// TIA Portal project "sauc" (V13)

(* hardware
DEVICE "HMI_1"  TP700 Comfort
   slot 0: "HMI"  HMI  6AV2 124-0GC01-0AX0  13.0.1.0
   slot 1: "HMI_RT_1"  TP700 Comfort  6AV2 124-0GC01-0AX0  13.0.1.0
   slot 5: "HMI_1.IE_CP_1"  PROFINET Interface
      slot 1: "PROFINET Interface_1"  PROFINET Interface
         slot 1: "Port_1"  Port
         slot 2: "Port_2"  Port
   slot 7: "HMI_1.MPI/DP_CP_1"  MPI/DP Interface
*)

(* ===== HMI "HMI_RT_1" =====
connection "CPU224": IF1 B, SIMATIC S7 200

HMI tags "Default tag table"
   "lightSensor" : Bool, 1 s
   "openDoor" : Bool, 1 s
   "lowBob" : Bool, 1 s
   "upBob" : Bool, 1 s
   "heaterGoOn" : Bool, 1 s
   "lightGoOn" : Bool, 1 s
   "doorGoOn" : Bool, 1 s
   "ventilGoOn" : Bool, 1 s
   "valve1goOn" : Bool, 1 s
   "valve2goOn" : Bool, 1 s
   "valve3goOn" : Bool, 1 s
   "lightBySensor" : Bool, 1 s
   "lightByTime" : Bool, 1 s
   "readYear" : Byte, 1 s
   "readMonth" : Byte, 1 s
   "readDay" : Byte, 1 s
   "readHours" : Byte, 1 s
   "readMinutes" : Byte, 1 s
   "readSeconds" : Byte, 1 s
   "writeYear" : Byte, 1 s
   "writeMonth" : Byte, 1 s
   "writeDay" : Byte, 1 s
   "writeHours" : Byte, 1 s
   "writeMinutes" : Byte, 1 s
   "writeSeconds" : Byte, 1 s
   "roomTemp4ma" : Real, 1 s
   "roomTemp20ma" : Real, 1 s
   "airTemp4ma" : Real, 1 s
   "airTemp20ma" : Real, 1 s
   "humidityRoom4ma" : Real, 1 s
   "humidityRoom20ma" : Real, 1 s
   "floorTemp4ma" : Real, 1 s
   "floorTemp20ma" : Real, 1 s
   "roomTemp" : Real, 1 s
   "airTemp" : Real, 1 s
   "humidityRoom" : Real, 1 s
   "floorTemp" : Real, 1 s
   "v1_e1_on_hh" : Byte, 1 s
   "v1_e1_on_mm" : Byte, 1 s
   "v1_e1_off_hh" : Byte, 1 s
   "v1_e1_off_mm" : Byte, 1 s
   "v1_e2_on_hh" : Byte, 1 s
   "v1_e2_on_mm" : Byte, 1 s
   "v1_e2_off_hh" : Byte, 1 s
   "v1_e2_off_mm" : Byte, 1 s
   "v1_e3_on_hh" : Byte, 1 s
   "v1_e3_on_mm" : Byte, 1 s
   "v1_e3_off_hh" : Byte, 1 s
   "v1_e3_off_mm" : Byte, 1 s
   "v1_e4_on_hh" : Byte, 1 s
   "v1_e4_on_mm" : Byte, 1 s
   "v1_e4_off_hh" : Byte, 1 s
   "v1_e4_off_mm" : Byte, 1 s
   "v1_e5_on_hh" : Byte, 1 s
   "v1_e5_on_mm" : Byte, 1 s
   "v1_e5_off_hh" : Byte, 1 s
   "v1_e5_off_mm" : Byte, 1 s
   "v2_e1_on_hh" : Byte, 1 s
   "v2_e1_on_mm" : Byte, 1 s
   "v2_e1_off_hh" : Byte, 1 s
   "v2_e1_off_mm" : Byte, 1 s
   "v2_e2_on_hh" : Byte, 1 s
   "v2_e2_on_mm" : Byte, 1 s
   "v2_e2_off_hh" : Byte, 1 s
   "v2_e2_off_mm" : Byte, 1 s
   "v2_e3_on_hh" : Byte, 1 s
   "v2_e3_on_mm" : Byte, 1 s
   "v2_e3_off_hh" : Byte, 1 s
   "v2_e3_off_mm" : Byte, 1 s
   "v2_e4_on_hh" : Byte, 1 s
   "v2_e4_on_mm" : Byte, 1 s
   "v2_e4_off_hh" : Byte, 1 s
   "v2_e4_off_mm" : Byte, 1 s
   "v2_e5_on_hh" : Byte, 1 s
   "v2_e5_on_mm" : Byte, 1 s
   "v2_e5_off_hh" : Byte, 1 s
   "v2_e5_off_mm" : Byte, 1 s
   "light_e1_on_hh" : Byte, 1 s
   "light_e1_on_mm" : Byte, 1 s
   "light_e1_off_hh" : Byte, 1 s
   "light_e1_off_mm" : Byte, 1 s
   "light_e2_on_hh" : Byte, 1 s
   "light_e2_on_mm" : Byte, 1 s
   "light_e2_off_hh" : Byte, 1 s
   "light_e2_off_mm" : Byte, 1 s
   "door_e1_on_hh" : Byte, 1 s
   "door_e1_on_mm" : Byte, 1 s
   "door_e1_off_hh" : Byte, 1 s
   "door_e1_off_mm" : Byte, 1 s
   "door_e2_on_hh" : Byte, 1 s
   "door_e2_on_mm" : Byte, 1 s
   "door_e2_off_hh" : Byte, 1 s
   "door_e2_off_mm" : Byte, 1 s
   "lowSpWithAir" : Real, 1 s
   "upSpWithAir" : Real, 1 s
   "lowSpWithFloor" : Real, 1 s
   "upSpWithFloor" : Real, 1 s
   "lightHandOn" : Bool, 1 s
   "lightHandOff" : Bool, 1 s
   "heatSensorIsAir" : Bool, 1 s
   "heatHandOn" : Bool, 1 s
   "heatHandOff" : Bool, 1 s
   "doorHandOn" : Bool, 1 s
   "doorHandOff" : Bool, 1 s
   "setClock" : Bool, 1 s
   "lightHandGo" : Bool, 1 s
   "doorHandGo" : Bool, 1 s
   "ventilSensorIsTemp" : Bool, 1 s
   "lowSpWithTemp" : Real, 1 s
   "upSpWithTemp" : Real, 1 s
   "lowSpWithHumi" : Real, 1 s
   "upSpWithHumi" : Real, 1 s
   "heat2goOn" : Bool, 1 s
   "lowSpWithOutside" : Real, 1 s
   "upSpWithOutside" : Real, 1 s
   "im1_e1_off_hh" : Byte, 1 s
   "im1_e1_off_mm" : Byte, 1 s
   "im1_e1_on_hh" : Byte, 1 s
   "im1_e1_on_mm" : Byte, 1 s
   "im1_e2_off_hh" : Byte, 1 s
   "im1_e2_off_mm" : Byte, 1 s
   "im1_e2_on_hh" : Byte, 1 s
   "im1_e2_on_mm" : Byte, 1 s
   "im1_e3_off_hh" : Byte, 1 s
   "im1_e3_off_mm" : Byte, 1 s
   "im1_e3_on_hh" : Byte, 1 s
   "im1_e3_on_mm" : Byte, 1 s
   "im1_e4_off_hh" : Byte, 1 s
   "im1_e4_off_mm" : Byte, 1 s
   "im1_e4_on_hh" : Byte, 1 s
   "im1_e4_on_mm" : Byte, 1 s
   "im1_e5_off_hh" : Byte, 1 s
   "im1_e5_off_mm" : Byte, 1 s
   "im1_e5_on_hh" : Byte, 1 s
   "im1_e5_on_mm" : Byte, 1 s
   "im2_e1_off_hh" : Byte, 1 s
   "im2_e1_off_mm" : Byte, 1 s
   "im2_e1_on_hh" : Byte, 1 s
   "im2_e1_on_mm" : Byte, 1 s
   "im2_e2_off_hh" : Byte, 1 s
   "im2_e2_off_mm" : Byte, 1 s
   "im2_e2_on_hh" : Byte, 1 s
   "im2_e2_on_mm" : Byte, 1 s
   "im2_e3_off_hh" : Byte, 1 s
   "im2_e3_off_mm" : Byte, 1 s
   "im2_e3_on_hh" : Byte, 1 s
   "im2_e3_on_mm" : Byte, 1 s
   "im2_e4_off_hh" : Byte, 1 s
   "im2_e4_off_mm" : Byte, 1 s
   "im2_e4_on_hh" : Byte, 1 s
   "im2_e4_on_mm" : Byte, 1 s
   "im2_e5_off_hh" : Byte, 1 s
   "im2_e5_off_mm" : Byte, 1 s
   "im2_e5_on_hh" : Byte, 1 s
   "im2_e5_on_mm" : Byte, 1 s
   "im1goOn" : Bool, 1 s
   "im2goOn" : Bool, 1 s
   "humidityMax" : Real, internal
   "humidityMin" : Real, internal
   "flowTotal" : DWord, 1 s
   "impulseWeight" : DWord, 1 s
   "resetFlow" : Bool, 1 s

screen "main" 800x480
   GraphicView "Graphic view_2" at 671,255 size 29x190
   GraphicView "Graphic view_1" at 630,142 size 107x173
   GraphicView "Graphic view_13" at 597,409 size 19x54
   GraphicIOField "Graphic I/O field_3" at 386,34 size 76x80
   GraphicIOField "Graphic I/O field_4" at 684,24 size 61x90
   GraphicIOField "Graphic I/O field_1" at 536,36 size 71x83
   Clock "Clock_1" at 326,157 size 174x167
   GraphicView "Graphic view_16" at 356,333 size 100x101
   GraphicView "Graphic view_11" at 613,287 size 30x26
   GraphicView "Graphic view_12" at 624,308 size 19x134
   GraphicView "Graphic view_10" at 510,286 size 107x18
   GraphicView "Graphic view_8" at 523,395 size 67x18
   GraphicView "Graphic view_6" at 693,357 size 29x35
   Gauge "Gauge_1" at 21,46 size 143x143
   TextField "Text field_1" at 639,172 size 64x18
   TextField "Text field_2" at 639,214 size 64x18
   TextField "Text field_3" at 47,7 size 110x21
   TextField "Text field_4" at 45,24 size 115x21
   IOField "I/O field_3" at 58,164 size 68x32
   TextField "Text field_13" at 377,12 size 105x21
   TextField "Text field_14" at 527,169 size 40x21
   TextField "Text field_16" at 516,12 size 120x21
   SymbolicIOField "Symbolic I/O field_2" at 399,116 size 57x20
   TextField "Text field_17" at 520,231 size 42x18
   SymbolicIOField "Symbolic I/O field_5" at 517,304 size 60x24
   TextField "Text field_18" at 511,341 size 76x18
   SymbolicIOField "Symbolic I/O field_7" at 711,383 size 59x24
   Button "Button_1" at 360,350 size 96x75
   Button "Button_2" at 498,364 size 104x54
   Button "Button_3" at 520,41 size 104x69
   Button "Button_4" at 508,153 size 81x59
   Button "Button_5" at 663,30 size 100x84
   Button "Button_6" at 345,186 size 132x113
   Button "Button_7" at 370,35 size 109x78
   TextField "Text field_21" at 639,187 size 64x18
   TextField "Text field_22" at 639,232 size 64x18
   GraphicView "Graphic view_3" at 512,254 size 46x52
   GraphicView "Graphic view_4" at 512,363 size 46x52
   GraphicView "Graphic view_5" at 705,327 size 52x58
   TextField "Text field_8" at 217,7 size 110x21
   IOField "I/O field_1" at 58,433 size 68x32
   TextField "Text field_5" at 243,24 size 45x21
   Gauge "Gauge_4" at 197,46 size 143x143
   IOField "I/O field_2" at 234,164 size 68x32
   TextField "Text field_6" at 21,210 size 189x21
   Bar "Bar_2" at 55,230 size 76x192
   TextField "Text field_11" at 127,439 size 24x21
   IOField "I/O field_4" at 237,433 size 68x32
   TextField "Text field_23" at 228,210 size 95x21
   Bar "Bar_1" at 233,230 size 76x192
   TextField "Text field_9" at 304,439 size 23x21
   GraphicView "Graphic view_7" at 569,429 size 156x45
   GraphicView "Graphic view_9" at 586,396 size 30x26
   Button "Button_8" at 495,255 size 104x54
   SymbolicIOField "Symbolic I/O field_6" at 518,418 size 58x24
   TextField "Text field_7" at 361,439 size 104x21
   Button "Button_9" at 685,331 size 104x54
   IOField "I/O field_5" at 703,407 size 83x20
   TextField "Text field_10" at 755,171 size 40x18
   TextField "Text field_12" at 755,230 size 40x18

screen "calibration" 800x480
   TextField "Text field_1" at 330,34 size 116x23
   TextField "Text field_2" at 43,115 size 127x23
   TextField "Text field_3" at 43,138 size 129x23
   TextField "Text field_4" at 237,114 size 127x23
   TextField "Text field_5" at 252,137 size 88x23
   TextField "Text field_6" at 451,112 size 106x23
   TextField "Text field_7" at 441,135 size 129x23
   TextField "Text field_8" at 637,110 size 127x23
   TextField "Text field_9" at 664,133 size 49x23
   TextField "Text field_10" at 30,199 size 48x23
   TextField "Text field_11" at 20,259 size 59x23
   TextField "Text field_12" at 234,197 size 48x23
   TextField "Text field_13" at 224,257 size 59x23
   TextField "Text field_14" at 450,195 size 48x23
   TextField "Text field_15" at 440,255 size 59x23
   TextField "Text field_16" at 633,196 size 48x23
   TextField "Text field_17" at 623,256 size 59x23
   IOField "I/O field_1" at 89,195 size 68x32
   IOField "I/O field_2" at 89,250 size 68x32
   IOField "I/O field_3" at 288,196 size 68x32
   IOField "I/O field_4" at 288,251 size 68x32
   IOField "I/O field_5" at 503,197 size 68x32
   IOField "I/O field_6" at 503,252 size 68x32
   IOField "I/O field_7" at 685,193 size 68x32
   IOField "I/O field_8" at 685,248 size 68x32
   TextField "Text field_18" at 159,199 size 26x23
   TextField "Text field_19" at 157,257 size 26x23
   TextField "Text field_20" at 357,199 size 26x23
   TextField "Text field_21" at 356,255 size 26x23
   TextField "Text field_22" at 755,199 size 26x23
   TextField "Text field_23" at 755,252 size 26x23
   TextField "Text field_24" at 573,197 size 25x23
   TextField "Text field_25" at 573,257 size 25x23
   Button "Button_1" at 14,16 size 117x33
   IOField "I/O field_9" at 58,363 size 68x32
   TextField "Text field_26" at 127,366 size 26x23
   TextField "Text field_27" at 44,308 size 88x23
   TextField "Text field_28" at 73,331 size 91x23
   IOField "I/O field_10" at 259,363 size 68x32
   TextField "Text field_29" at 328,366 size 26x23
   TextField "Text field_30" at 245,308 size 88x23
   TextField "Text field_31" at 274,331 size 91x23
   IOField "I/O field_11" at 460,363 size 68x32
   TextField "Text field_32" at 529,366 size 25x23
   TextField "Text field_33" at 446,308 size 88x23
   TextField "Text field_34" at 475,331 size 91x23
   IOField "I/O field_12" at 661,363 size 68x32
   TextField "Text field_35" at 730,366 size 26x23
   TextField "Text field_36" at 647,308 size 88x23
   TextField "Text field_37" at 676,331 size 91x23

screen "valves" 800x480
   TextField "Text field_1" at 184,43 size 89x23
   TextField "Text field_26" at 545,43 size 89x23
   TextField "Text field_27" at 66,132 size 30x23
   TextField "Text field_28" at 66,205 size 30x23
   TextField "Text field_29" at 66,278 size 30x23
   TextField "Text field_30" at 66,351 size 30x23
   TextField "Text field_31" at 66,424 size 30x23
   Button "Button_1" at 14,16 size 117x33
   IOField "I/O field_21" at 108,129 size 32x32
   IOField "I/O field_22" at 155,129 size 32x32
   TextField "Text field_14" at 142,135 size 12x23
   IOField "I/O field_23" at 273,129 size 32x32
   IOField "I/O field_24" at 320,129 size 32x32
   TextField "Text field_15" at 307,135 size 12x23
   IOField "I/O field_25" at 108,201 size 32x32
   IOField "I/O field_26" at 155,201 size 32x32
   TextField "Text field_16" at 142,207 size 12x23
   IOField "I/O field_27" at 273,201 size 32x32
   IOField "I/O field_28" at 320,201 size 32x32
   TextField "Text field_17" at 307,207 size 12x23
   IOField "I/O field_29" at 108,273 size 32x32
   IOField "I/O field_30" at 155,273 size 32x32
   TextField "Text field_18" at 142,279 size 12x23
   IOField "I/O field_31" at 273,273 size 32x32
   IOField "I/O field_32" at 320,273 size 32x32
   TextField "Text field_19" at 307,279 size 12x23
   IOField "I/O field_33" at 108,345 size 32x32
   IOField "I/O field_34" at 155,345 size 32x32
   TextField "Text field_20" at 142,351 size 12x23
   IOField "I/O field_35" at 273,345 size 32x32
   IOField "I/O field_36" at 320,345 size 32x32
   TextField "Text field_21" at 307,351 size 12x23
   IOField "I/O field_37" at 108,417 size 32x32
   IOField "I/O field_38" at 155,417 size 32x32
   TextField "Text field_22" at 142,423 size 12x23
   IOField "I/O field_39" at 273,417 size 32x32
   IOField "I/O field_40" at 320,417 size 32x32
   TextField "Text field_23" at 307,423 size 12x23
   TextField "Text field_24" at 97,88 size 110x23
   TextField "Text field_25" at 251,86 size 121x23
   IOField "I/O field_3" at 458,129 size 32x32
   IOField "I/O field_1" at 505,129 size 32x32
   TextField "Text field_2" at 492,135 size 12x23
   IOField "I/O field_2" at 623,129 size 32x32
   IOField "I/O field_4" at 670,129 size 32x32
   TextField "Text field_3" at 657,135 size 12x23
   IOField "I/O field_5" at 458,201 size 32x32
   IOField "I/O field_6" at 505,201 size 32x32
   TextField "Text field_4" at 492,207 size 12x23
   IOField "I/O field_7" at 623,201 size 32x32
   IOField "I/O field_8" at 670,201 size 32x32
   TextField "Text field_5" at 657,207 size 12x23
   IOField "I/O field_9" at 458,273 size 32x32
   IOField "I/O field_10" at 505,273 size 32x32
   TextField "Text field_6" at 492,279 size 12x23
   IOField "I/O field_11" at 623,273 size 32x32
   IOField "I/O field_12" at 670,273 size 32x32
   TextField "Text field_7" at 657,279 size 12x23
   IOField "I/O field_13" at 458,345 size 32x32
   IOField "I/O field_14" at 505,345 size 32x32
   TextField "Text field_8" at 492,351 size 12x23
   IOField "I/O field_15" at 623,345 size 32x32
   IOField "I/O field_16" at 670,345 size 32x32
   TextField "Text field_9" at 657,351 size 12x23
   IOField "I/O field_17" at 458,417 size 32x32
   IOField "I/O field_18" at 505,417 size 32x32
   TextField "Text field_10" at 492,423 size 12x23
   IOField "I/O field_19" at 623,417 size 32x32
   IOField "I/O field_20" at 670,417 size 32x32
   TextField "Text field_11" at 657,423 size 12x23
   TextField "Text field_12" at 447,88 size 110x23
   TextField "Text field_13" at 601,86 size 121x23
   Button "Button_2" at 663,16 size 117x33

screen "heater" 800x480
   TextField "Text field_1" at 373,28 size 82x23
   Button "Button_1" at 14,16 size 117x33
   Switch "Switch_1" at 291,123 size 216x82
   IOField "I/O field_21" at 107,299 size 67x32
   TextField "Text field_24" at 65,273 size 149x23
   TextField "Text field_25" at 54,360 size 160x23
   TextField "Text field_3" at 87,86 size 127x23
   TextField "Text field_4" at 104,109 size 80x23
   IOField "I/O field_3" at 106,151 size 68x32
   TextField "Text field_20" at 175,154 size 26x23
   TextField "Text field_2" at 175,303 size 26x23
   IOField "I/O field_1" at 107,392 size 67x32
   TextField "Text field_5" at 175,396 size 26x23
   TextField "Text field_9" at 593,86 size 127x23
   TextField "Text field_10" at 631,109 size 49x23
   IOField "I/O field_2" at 618,151 size 68x32
   TextField "Text field_12" at 687,154 size 26x23
   IOField "I/O field_4" at 619,299 size 67x32
   TextField "Text field_6" at 577,273 size 149x23
   TextField "Text field_7" at 566,360 size 160x23
   TextField "Text field_8" at 687,303 size 26x23
   IOField "I/O field_5" at 619,392 size 67x32
   TextField "Text field_11" at 687,396 size 26x23
   TextField "Text field_13" at 296,259 size 237x23
   SymbolicIOField "Symbolic I/O field_1" at 380,416 size 73x23
   Button "Button_2" at 617,16 size 162x33

screen "light" 800x480
   Button "Button_1" at 14,16 size 117x33
   TextField "Text field_27" at 372,131 size 30x23
   TextField "Text field_28" at 372,204 size 30x23
   IOField "I/O field_21" at 414,128 size 32x32
   IOField "I/O field_22" at 461,128 size 32x32
   TextField "Text field_14" at 448,134 size 12x23
   IOField "I/O field_23" at 579,128 size 32x32
   IOField "I/O field_24" at 626,128 size 32x32
   TextField "Text field_15" at 613,134 size 12x23
   IOField "I/O field_25" at 414,200 size 32x32
   IOField "I/O field_26" at 461,200 size 32x32
   TextField "Text field_16" at 448,206 size 12x23
   IOField "I/O field_27" at 579,200 size 32x32
   IOField "I/O field_28" at 626,200 size 32x32
   TextField "Text field_17" at 613,206 size 12x23
   TextField "Text field_24" at 403,87 size 110x23
   TextField "Text field_25" at 557,85 size 121x23
   TextField "Text field_1" at 338,31 size 110x23
   TextField "Text field_13" at 529,265 size 211x23
   SymbolicIOField "Symbolic I/O field_1" at 577,417 size 116x23
   Switch "Switch_1" at 62,115 size 184x88
   Switch "Switch_2" at 62,305 size 184x88
   Switch "Switch_3" at 316,305 size 184x88

screen "door" 800x480
   Button "Button_1" at 14,16 size 117x33
   TextField "Text field_27" at 152,129 size 30x23
   TextField "Text field_28" at 152,202 size 30x23
   IOField "I/O field_21" at 194,126 size 32x32
   IOField "I/O field_22" at 241,126 size 32x32
   TextField "Text field_14" at 228,132 size 12x23
   IOField "I/O field_23" at 359,126 size 32x32
   IOField "I/O field_24" at 406,126 size 32x32
   TextField "Text field_15" at 393,132 size 12x23
   IOField "I/O field_25" at 194,198 size 32x32
   IOField "I/O field_26" at 241,198 size 32x32
   TextField "Text field_16" at 228,204 size 12x23
   IOField "I/O field_27" at 359,198 size 32x32
   IOField "I/O field_28" at 406,198 size 32x32
   TextField "Text field_17" at 393,204 size 12x23
   TextField "Text field_24" at 183,85 size 96x23
   TextField "Text field_25" at 345,83 size 95x23
   TextField "Text field_1" at 376,28 size 61x23
   TextField "Text field_13" at 302,274 size 164x23
   SymbolicIOField "Symbolic I/O field_1" at 338,426 size 116x23
   Switch "Switch_3" at 522,116 size 184x88

screen "clock" 800x480
   TextField "Text field_1" at 358,26 size 63x23
   IOField "I/O field_21" at 346,289 size 31x32
   TextField "Text field_2" at 379,293 size 12x23
   IOField "I/O field_1" at 393,289 size 31x32
   IOField "I/O field_2" at 306,353 size 31x32
   TextField "Text field_3" at 342,362 size 11x23
   IOField "I/O field_3" at 357,353 size 31x32
   TextField "Text field_4" at 396,362 size 11x23
   IOField "I/O field_4" at 414,353 size 31x32
   Button "Button_1" at 14,16 size 117x33
   Button "Button_2" at 322,410 size 117x33
   IOField "I/O field_9" at 199,115 size 35x32
   TextField "Text field_5" at 238,118 size 13x26
   IOField "I/O field_5" at 254,115 size 35x32
   TextField "Text field_6" at 294,118 size 13x26
   IOField "I/O field_6" at 312,115 size 35x32
   IOField "I/O field_7" at 404,115 size 35x32
   TextField "Text field_7" at 442,121 size 12x26
   IOField "I/O field_8" at 456,115 size 35x32
   IOField "I/O field_10" at 508,115 size 35x32
   TextField "Text field_8" at 493,121 size 12x26
   TextField "Text field_9" at 337,232 size 103x23

screen "ventil" 800x480
   TextField "Text field_1" at 352,28 size 116x23
   Button "Button_1" at 14,16 size 117x33
   Switch "Switch_1" at 276,127 size 252x82
   IOField "I/O field_21" at 86,299 size 88x32
   TextField "Text field_24" at 65,273 size 149x23
   TextField "Text field_25" at 54,360 size 160x23
   TextField "Text field_3" at 75,86 size 127x23
   TextField "Text field_4" at 92,109 size 80x23
   IOField "I/O field_3" at 82,151 size 92x32
   TextField "Text field_20" at 175,154 size 26x23
   TextField "Text field_2" at 175,303 size 26x23
   IOField "I/O field_1" at 85,392 size 89x32
   TextField "Text field_5" at 175,396 size 26x23
   TextField "Text field_9" at 601,90 size 106x23
   IOField "I/O field_2" at 603,151 size 91x32
   TextField "Text field_12" at 695,154 size 25x23
   IOField "I/O field_4" at 605,299 size 89x32
   TextField "Text field_6" at 580,273 size 149x23
   TextField "Text field_7" at 570,360 size 160x23
   TextField "Text field_8" at 695,303 size 25x23
   IOField "I/O field_5" at 607,392 size 87x32
   TextField "Text field_11" at 695,396 size 25x23
   TextField "Text field_13" at 304,259 size 218x23
   SymbolicIOField "Symbolic I/O field_1" at 382,416 size 73x23

screen "heater2" 800x480
   TextField "Text field_1" at 299,27 size 230x23
   Button "Button_1" at 14,16 size 117x33
   IOField "I/O field_21" at 153,300 size 89x32
   TextField "Text field_24" at 133,274 size 149x23
   TextField "Text field_25" at 122,361 size 160x23
   TextField "Text field_3" at 303,122 size 216x23
   IOField "I/O field_3" at 341,163 size 91x32
   TextField "Text field_20" at 436,166 size 26x23
   TextField "Text field_2" at 243,304 size 26x23
   IOField "I/O field_1" at 154,393 size 88x32
   TextField "Text field_5" at 243,397 size 26x23
   TextField "Text field_13" at 490,254 size 237x23
   SymbolicIOField "Symbolic I/O field_1" at 569,411 size 73x23

screen "ims" 800x480
   TextField "Text field_1" at 175,43 size 50x23
   TextField "Text field_26" at 553,43 size 50x23
   TextField "Text field_27" at 57,132 size 30x23
   TextField "Text field_28" at 57,205 size 30x23
   TextField "Text field_29" at 57,278 size 30x23
   TextField "Text field_30" at 57,351 size 30x23
   TextField "Text field_31" at 57,424 size 30x23
   Button "Button_1" at 14,16 size 117x33
   IOField "I/O field_21" at 99,129 size 32x32
   IOField "I/O field_22" at 146,129 size 32x32
   TextField "Text field_14" at 133,135 size 12x23
   IOField "I/O field_23" at 264,129 size 32x32
   IOField "I/O field_24" at 311,129 size 32x32
   TextField "Text field_15" at 298,135 size 12x23
   IOField "I/O field_25" at 99,201 size 32x32
   IOField "I/O field_26" at 146,201 size 32x32
   TextField "Text field_16" at 133,207 size 12x23
   IOField "I/O field_27" at 264,201 size 32x32
   IOField "I/O field_28" at 311,201 size 32x32
   TextField "Text field_17" at 298,207 size 12x23
   IOField "I/O field_29" at 99,273 size 32x32
   IOField "I/O field_30" at 146,273 size 32x32
   TextField "Text field_18" at 133,279 size 12x23
   IOField "I/O field_31" at 264,273 size 32x32
   IOField "I/O field_32" at 311,273 size 32x32
   TextField "Text field_19" at 298,279 size 12x23
   IOField "I/O field_33" at 99,345 size 32x32
   IOField "I/O field_34" at 146,345 size 32x32
   TextField "Text field_20" at 133,351 size 12x23
   IOField "I/O field_35" at 264,345 size 32x32
   IOField "I/O field_36" at 311,345 size 32x32
   TextField "Text field_21" at 298,351 size 12x23
   IOField "I/O field_37" at 99,417 size 32x32
   IOField "I/O field_38" at 146,417 size 32x32
   TextField "Text field_22" at 133,423 size 12x23
   IOField "I/O field_39" at 264,417 size 32x32
   IOField "I/O field_40" at 311,417 size 32x32
   TextField "Text field_23" at 298,423 size 12x23
   TextField "Text field_24" at 88,88 size 110x23
   TextField "Text field_25" at 242,86 size 121x23
   IOField "I/O field_3" at 466,129 size 32x32
   IOField "I/O field_1" at 513,129 size 32x32
   TextField "Text field_2" at 500,135 size 12x23
   IOField "I/O field_2" at 631,129 size 32x32
   IOField "I/O field_4" at 678,129 size 32x32
   TextField "Text field_3" at 665,135 size 12x23
   IOField "I/O field_5" at 466,201 size 32x32
   IOField "I/O field_6" at 513,201 size 32x32
   TextField "Text field_4" at 500,207 size 12x23
   IOField "I/O field_7" at 631,201 size 32x32
   IOField "I/O field_8" at 678,201 size 32x32
   TextField "Text field_5" at 665,207 size 12x23
   IOField "I/O field_9" at 466,273 size 32x32
   IOField "I/O field_10" at 513,273 size 32x32
   TextField "Text field_6" at 500,279 size 12x23
   IOField "I/O field_11" at 631,273 size 32x32
   IOField "I/O field_12" at 678,273 size 32x32
   TextField "Text field_7" at 665,279 size 12x23
   IOField "I/O field_13" at 466,345 size 32x32
   IOField "I/O field_14" at 513,345 size 32x32
   TextField "Text field_8" at 500,351 size 12x23
   IOField "I/O field_15" at 631,345 size 32x32
   IOField "I/O field_16" at 678,345 size 32x32
   TextField "Text field_9" at 665,351 size 12x23
   IOField "I/O field_17" at 466,417 size 32x32
   IOField "I/O field_18" at 513,417 size 32x32
   TextField "Text field_10" at 500,423 size 12x23
   IOField "I/O field_19" at 631,417 size 32x32
   IOField "I/O field_20" at 678,417 size 32x32
   TextField "Text field_11" at 665,423 size 12x23
   TextField "Text field_12" at 455,88 size 110x23
   TextField "Text field_13" at 609,86 size 121x23

screen "flow" 800x480
   Button "Button_1" at 14,16 size 117x33
   TextField "Text field_1" at 376,28 size 71x23
   TextField "Text field_3" at 69,119 size 140x23
   IOField "I/O field_3" at 67,151 size 126x32
   TextField "Text field_20" at 200,155 size 16x23
   TextField "Text field_2" at 290,118 size 129x23
   IOField "I/O field_1" at 301,150 size 63x32
   TextField "Text field_4" at 367,155 size 16x23
   Button "Button_2" at 71,204 size 117x33
*)